// TIA Portal V17 export
// export: Created 2022-07-20T06:59:48.5903746Z, ExportSetting WithDefaults, DisplayName Totally Integrated Automation Portal, DisplayVersion V17, DisplayName TIA Portal Openness, DisplayVersion V17, DisplayName TIA Portal Version Control Interface, DisplayVersion V17, DisplayName SINAMICS Startdrive Advanced, DisplayVersion V17, DisplayName SINAMICS Startdrive G130, G150, S120, S150, SINAMICS MV, S210, DisplayVersion V17, DisplayName SINAMICS Startdrive G110M, G120, G120C, G120D, G120P, G115D, DisplayVersion V17, DisplayName STEP 7 Professional, DisplayVersion V17, DisplayName STEP 7 Safety, DisplayVersion V17, DisplayName WinCC Advanced, DisplayVersion V17
FUNCTION_BLOCK "FB10210_SheetSolenoidValveManager"   // FB10210, LAD
TITLE = FB10210_SheetSolenoidValveManager
{ S7_Optimized_Access := 'TRUE' }
AUTHOR : Anirouddh
FAMILY : 1021x_SOLENOID_VALVES
VERSION : 1.0
// Release note : 
// 1.0 - Feature developped
// stored: AutoNumber false, IsIECCheckEnabled false, IsRetainMemResEnabled false, MemoryReserve 100, SetENOAutomatically false, UDAEnableTagReadback false
   VAR_INPUT
      OptionManageSolenoidValve : Bool;
      RequestActiveSolenoidValve : Bool;
   END_VAR
   VAR_OUTPUT
      ActiveSoleinoidValve : Bool;
   END_VAR
BEGIN

REGION Network 1 (SCL)
   IF #OptionManageSolenoidValve AND #RequestActiveSolenoidValve THEN
       #ActiveSoleinoidValve := TRUE;
   ELSE
       #ActiveSoleinoidValve := FALSE;
   END_IF;
END_REGION
END_FUNCTION_BLOCK
